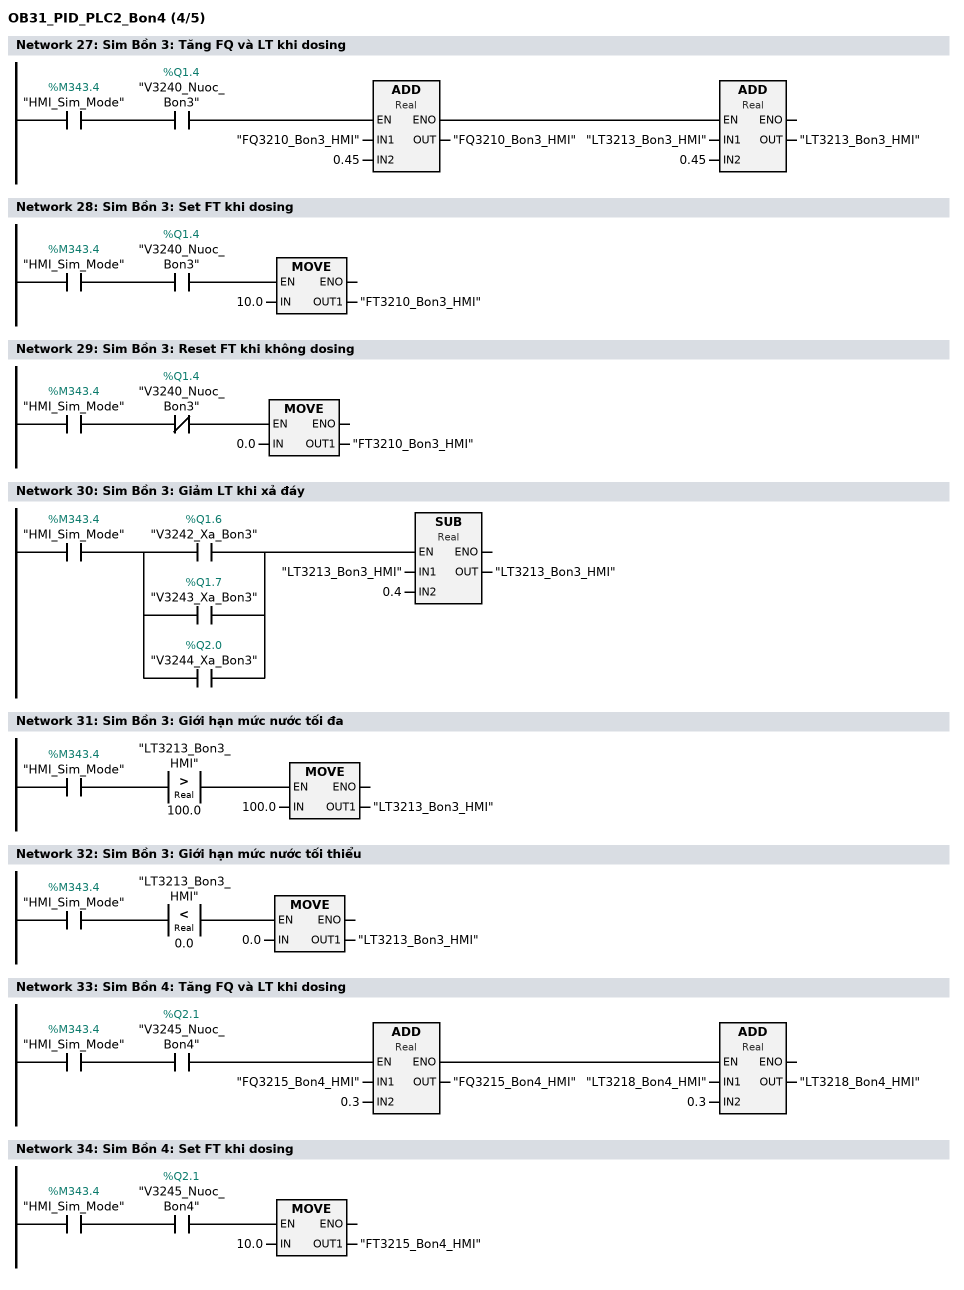
   RUNG wire#powerrail
      Contact( "HMI_Sim_Mode" )
      Contact( "V3240_Nuoc_Bon3" )
      { S7_Templates := "SrcType := Real"; S7_GenerateENO := "TRUE" } Add(in1 := "FQ3210_Bon3_HMI", in2 := 0.45, out => "FQ3210_Bon3_HMI")
      { S7_Templates := "SrcType := Real"; S7_GenerateENO := "TRUE" } Add(in1 := "LT3213_Bon3_HMI", in2 := 0.45, out => "LT3213_Bon3_HMI")
   END_RUNG
   // the same network as SCL:
   // ENO of a box is taken as its EN; it also drops when the box reports an error
   IF "HMI_Sim_Mode" AND "V3240_Nuoc_Bon3" THEN
       "FQ3210_Bon3_HMI" := "FQ3210_Bon3_HMI" + 0.45;
       "LT3213_Bon3_HMI" := "LT3213_Bon3_HMI" + 0.45;
   END_IF;
END_REGION

REGION Network 28: Sim Bồn 3: Set FT khi dosing
   RUNG wire#powerrail
      Contact( "HMI_Sim_Mode" )
      Contact( "V3240_Nuoc_Bon3" )
      { S7_GenerateENO := "TRUE" } Move(in := 10.0, out1 => "FT3210_Bon3_HMI")
   END_RUNG
   // the same network as SCL:
   IF "HMI_Sim_Mode" AND "V3240_Nuoc_Bon3" THEN "FT3210_Bon3_HMI" := 10.0; END_IF;
END_REGION

REGION Network 29: Sim Bồn 3: Reset FT khi không dosing
   RUNG wire#powerrail
      Contact( "HMI_Sim_Mode" )
      I_Contact( "V3240_Nuoc_Bon3" )
      { S7_GenerateENO := "TRUE" } Move(in := 0.0, out1 => "FT3210_Bon3_HMI")
   END_RUNG
   // the same network as SCL:
   IF "HMI_Sim_Mode" AND NOT "V3240_Nuoc_Bon3" THEN "FT3210_Bon3_HMI" := 0.0; END_IF;
END_REGION

REGION Network 30: Sim Bồn 3: Giảm LT khi xả đáy
   RUNG wire#powerrail
      Contact( "HMI_Sim_Mode" )
      wire#w1
      Contact( "V3242_Xa_Bon3" )
      wire#w2
      { S7_Templates := "SrcType := Real"; S7_GenerateENO := "TRUE" } Sub(in1 := "LT3213_Bon3_HMI", in2 := 0.4, out => "LT3213_Bon3_HMI")
   END_RUNG
   RUNG wire#w1
      Contact( "V3243_Xa_Bon3" )
   END_RUNG wire#w2
   RUNG wire#w1
      Contact( "V3244_Xa_Bon3" )
   END_RUNG wire#w2
   // the same network as SCL:
   IF "HMI_Sim_Mode" AND ("V3242_Xa_Bon3" OR "V3243_Xa_Bon3" OR "V3244_Xa_Bon3") THEN
       "LT3213_Bon3_HMI" := "LT3213_Bon3_HMI" - 0.4;
   END_IF;
END_REGION

REGION Network 31: Sim Bồn 3: Giới hạn mức nước tối đa
   RUNG wire#powerrail
      Contact( "HMI_Sim_Mode" )
      { S7_Templates := "SrcType := Real" } GT_Contact(in1 := "LT3213_Bon3_HMI", in2 := 100.0)
      { S7_GenerateENO := "TRUE" } Move(in := 100.0, out1 => "LT3213_Bon3_HMI")
   END_RUNG
   // the same network as SCL:
   IF "HMI_Sim_Mode" AND ("LT3213_Bon3_HMI" > 100.0) THEN "LT3213_Bon3_HMI" := 100.0; END_IF;
END_REGION

REGION Network 32: Sim Bồn 3: Giới hạn mức nước tối thiểu
   RUNG wire#powerrail
      Contact( "HMI_Sim_Mode" )
      { S7_Templates := "SrcType := Real" } LT_Contact(in1 := "LT3213_Bon3_HMI", in2 := 0.0)
      { S7_GenerateENO := "TRUE" } Move(in := 0.0, out1 => "LT3213_Bon3_HMI")
   END_RUNG
   // the same network as SCL:
   IF "HMI_Sim_Mode" AND ("LT3213_Bon3_HMI" < 0.0) THEN "LT3213_Bon3_HMI" := 0.0; END_IF;
END_REGION

REGION Network 33: Sim Bồn 4: Tăng FQ và LT khi dosing
   RUNG wire#powerrail
      Contact( "HMI_Sim_Mode" )
      Contact( "V3245_Nuoc_Bon4" )
      { S7_Templates := "SrcType := Real"; S7_GenerateENO := "TRUE" } Add(in1 := "FQ3215_Bon4_HMI", in2 := 0.3, out => "FQ3215_Bon4_HMI")
      { S7_Templates := "SrcType := Real"; S7_GenerateENO := "TRUE" } Add(in1 := "LT3218_Bon4_HMI", in2 := 0.3, out => "LT3218_Bon4_HMI")
   END_RUNG
   // the same network as SCL:
   // ENO of a box is taken as its EN; it also drops when the box reports an error
   IF "HMI_Sim_Mode" AND "V3245_Nuoc_Bon4" THEN
       "FQ3215_Bon4_HMI" := "FQ3215_Bon4_HMI" + 0.3;
       "LT3218_Bon4_HMI" := "LT3218_Bon4_HMI" + 0.3;
   END_IF;
END_REGION

REGION Network 34: Sim Bồn 4: Set FT khi dosing
   RUNG wire#powerrail
      Contact( "HMI_Sim_Mode" )
      Contact( "V3245_Nuoc_Bon4" )
      { S7_GenerateENO := "TRUE" } Move(in := 10.0, out1 => "FT3215_Bon4_HMI")
   END_RUNG
   // the same network as SCL:
   IF "HMI_Sim_Mode" AND "V3245_Nuoc_Bon4" THEN "FT3215_Bon4_HMI" := 10.0; END_IF;
END_REGION

REGION Network 35: Sim Bồn 4: Reset FT khi không dosing
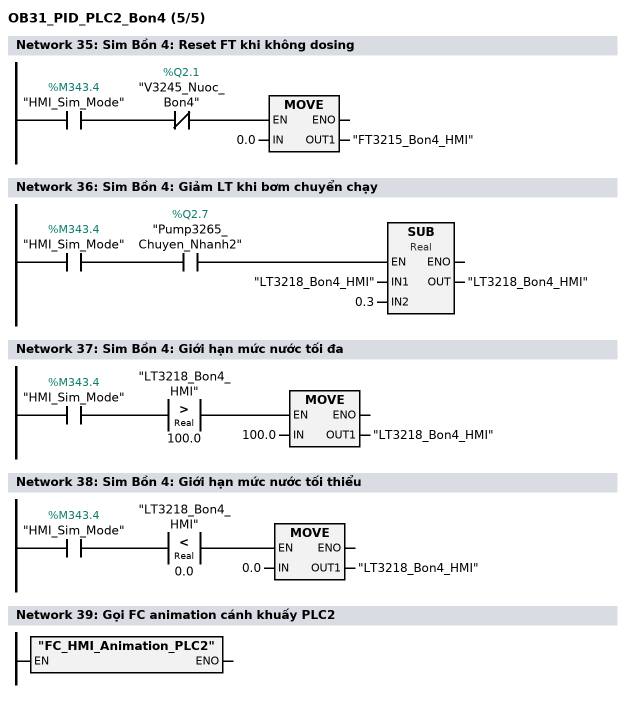
   RUNG wire#powerrail
      Contact( "HMI_Sim_Mode" )
      I_Contact( "V3245_Nuoc_Bon4" )
      { S7_GenerateENO := "TRUE" } Move(in := 0.0, out1 => "FT3215_Bon4_HMI")
   END_RUNG
   // the same network as SCL:
   IF "HMI_Sim_Mode" AND NOT "V3245_Nuoc_Bon4" THEN "FT3215_Bon4_HMI" := 0.0; END_IF;
END_REGION

REGION Network 36: Sim Bồn 4: Giảm LT khi bơm chuyển chạy
   RUNG wire#powerrail
      Contact( "HMI_Sim_Mode" )
      Contact( "Pump3265_Chuyen_Nhanh2" )
      { S7_Templates := "SrcType := Real"; S7_GenerateENO := "TRUE" } Sub(in1 := "LT3218_Bon4_HMI", in2 := 0.3, out => "LT3218_Bon4_HMI")
   END_RUNG
   // the same network as SCL:
   IF "HMI_Sim_Mode" AND "Pump3265_Chuyen_Nhanh2" THEN "LT3218_Bon4_HMI" := "LT3218_Bon4_HMI" - 0.3; END_IF;
END_REGION

REGION Network 37: Sim Bồn 4: Giới hạn mức nước tối đa
   RUNG wire#powerrail
      Contact( "HMI_Sim_Mode" )
      { S7_Templates := "SrcType := Real" } GT_Contact(in1 := "LT3218_Bon4_HMI", in2 := 100.0)
      { S7_GenerateENO := "TRUE" } Move(in := 100.0, out1 => "LT3218_Bon4_HMI")
   END_RUNG
   // the same network as SCL:
   IF "HMI_Sim_Mode" AND ("LT3218_Bon4_HMI" > 100.0) THEN "LT3218_Bon4_HMI" := 100.0; END_IF;
END_REGION

REGION Network 38: Sim Bồn 4: Giới hạn mức nước tối thiểu
   RUNG wire#powerrail
      Contact( "HMI_Sim_Mode" )
      { S7_Templates := "SrcType := Real" } LT_Contact(in1 := "LT3218_Bon4_HMI", in2 := 0.0)
      { S7_GenerateENO := "TRUE" } Move(in := 0.0, out1 => "LT3218_Bon4_HMI")
   END_RUNG
   // the same network as SCL:
   IF "HMI_Sim_Mode" AND ("LT3218_Bon4_HMI" < 0.0) THEN "LT3218_Bon4_HMI" := 0.0; END_IF;
END_REGION

REGION Network 39: Gọi FC animation cánh khuấy PLC2
   RUNG wire#powerrail
      "FC_HMI_Animation_PLC2"()
   END_RUNG
   // the same network as SCL:
   "FC_HMI_Animation_PLC2"();
END_REGION
END_ORGANIZATION_BLOCK

FUNCTION "FC_HMI_Animation_PLC2" : Void   // FC61, LAD
{ S7_Optimized_Access := 'TRUE' }
VERSION : 0.1
// stored: AutoNumber true, IsIECCheckEnabled false, SetENOAutomatically false, UDAEnableTagReadback false
BEGIN

REGION Network 1: Cánh khuấy Bồn 3: Tăng khung hình khi chạy
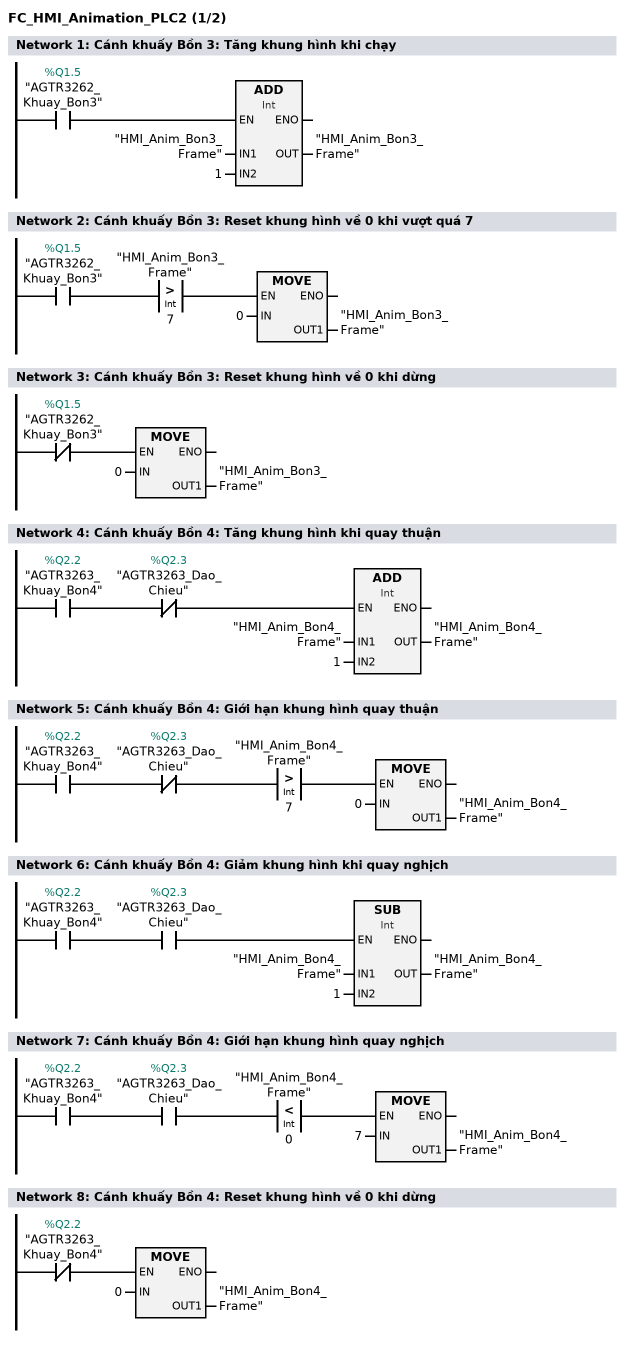
   RUNG wire#powerrail
      Contact( "AGTR3262_Khuay_Bon3" )
      { S7_Templates := "SrcType := Int"; S7_GenerateENO := "TRUE" } Add(in1 := "HMI_Anim_Bon3_Frame", in2 := 1, out => "HMI_Anim_Bon3_Frame")
   END_RUNG
   // the same network as SCL:
   IF "AGTR3262_Khuay_Bon3" THEN "HMI_Anim_Bon3_Frame" := "HMI_Anim_Bon3_Frame" + 1; END_IF;
END_REGION

REGION Network 2: Cánh khuấy Bồn 3: Reset khung hình về 0 khi vượt quá 7
   RUNG wire#powerrail
      Contact( "AGTR3262_Khuay_Bon3" )
      { S7_Templates := "SrcType := Int" } GT_Contact(in1 := "HMI_Anim_Bon3_Frame", in2 := 7)
      { S7_GenerateENO := "TRUE" } Move(in := 0, out1 => "HMI_Anim_Bon3_Frame")
   END_RUNG
   // the same network as SCL:
   IF "AGTR3262_Khuay_Bon3" AND ("HMI_Anim_Bon3_Frame" > 7) THEN "HMI_Anim_Bon3_Frame" := 0; END_IF;
END_REGION

REGION Network 3: Cánh khuấy Bồn 3: Reset khung hình về 0 khi dừng
   RUNG wire#powerrail
      I_Contact( "AGTR3262_Khuay_Bon3" )
      { S7_GenerateENO := "TRUE" } Move(in := 0, out1 => "HMI_Anim_Bon3_Frame")
   END_RUNG
   // the same network as SCL:
   IF NOT "AGTR3262_Khuay_Bon3" THEN "HMI_Anim_Bon3_Frame" := 0; END_IF;
END_REGION

REGION Network 4: Cánh khuấy Bồn 4: Tăng khung hình khi quay thuận
   RUNG wire#powerrail
      Contact( "AGTR3263_Khuay_Bon4" )
      I_Contact( "AGTR3263_Dao_Chieu" )
      { S7_Templates := "SrcType := Int"; S7_GenerateENO := "TRUE" } Add(in1 := "HMI_Anim_Bon4_Frame", in2 := 1, out => "HMI_Anim_Bon4_Frame")
   END_RUNG
   // the same network as SCL:
   IF "AGTR3263_Khuay_Bon4" AND NOT "AGTR3263_Dao_Chieu" THEN
       "HMI_Anim_Bon4_Frame" := "HMI_Anim_Bon4_Frame" + 1;
   END_IF;
END_REGION

REGION Network 5: Cánh khuấy Bồn 4: Giới hạn khung hình quay thuận
   RUNG wire#powerrail
      Contact( "AGTR3263_Khuay_Bon4" )
      I_Contact( "AGTR3263_Dao_Chieu" )
      { S7_Templates := "SrcType := Int" } GT_Contact(in1 := "HMI_Anim_Bon4_Frame", in2 := 7)
      { S7_GenerateENO := "TRUE" } Move(in := 0, out1 => "HMI_Anim_Bon4_Frame")
   END_RUNG
   // the same network as SCL:
   IF "AGTR3263_Khuay_Bon4" AND NOT "AGTR3263_Dao_Chieu" AND ("HMI_Anim_Bon4_Frame" > 7) THEN
       "HMI_Anim_Bon4_Frame" := 0;
   END_IF;
END_REGION

REGION Network 6: Cánh khuấy Bồn 4: Giảm khung hình khi quay nghịch
   RUNG wire#powerrail
      Contact( "AGTR3263_Khuay_Bon4" )
      Contact( "AGTR3263_Dao_Chieu" )
      { S7_Templates := "SrcType := Int"; S7_GenerateENO := "TRUE" } Sub(in1 := "HMI_Anim_Bon4_Frame", in2 := 1, out => "HMI_Anim_Bon4_Frame")
   END_RUNG
   // the same network as SCL:
   IF "AGTR3263_Khuay_Bon4" AND "AGTR3263_Dao_Chieu" THEN
       "HMI_Anim_Bon4_Frame" := "HMI_Anim_Bon4_Frame" - 1;
   END_IF;
END_REGION

REGION Network 7: Cánh khuấy Bồn 4: Giới hạn khung hình quay nghịch
   RUNG wire#powerrail
      Contact( "AGTR3263_Khuay_Bon4" )
      Contact( "AGTR3263_Dao_Chieu" )
      { S7_Templates := "SrcType := Int" } LT_Contact(in1 := "HMI_Anim_Bon4_Frame", in2 := 0)
      { S7_GenerateENO := "TRUE" } Move(in := 7, out1 => "HMI_Anim_Bon4_Frame")
   END_RUNG
   // the same network as SCL:
   IF "AGTR3263_Khuay_Bon4" AND "AGTR3263_Dao_Chieu" AND ("HMI_Anim_Bon4_Frame" < 0) THEN
       "HMI_Anim_Bon4_Frame" := 7;
   END_IF;
END_REGION

REGION Network 8: Cánh khuấy Bồn 4: Reset khung hình về 0 khi dừng
   RUNG wire#powerrail
      I_Contact( "AGTR3263_Khuay_Bon4" )
      { S7_GenerateENO := "TRUE" } Move(in := 0, out1 => "HMI_Anim_Bon4_Frame")
   END_RUNG
   // the same network as SCL:
   IF NOT "AGTR3263_Khuay_Bon4" THEN "HMI_Anim_Bon4_Frame" := 0; END_IF;
END_REGION

REGION Network 9: Bồn 3 Mức dịch: Rỗng khi LT <= 0.5
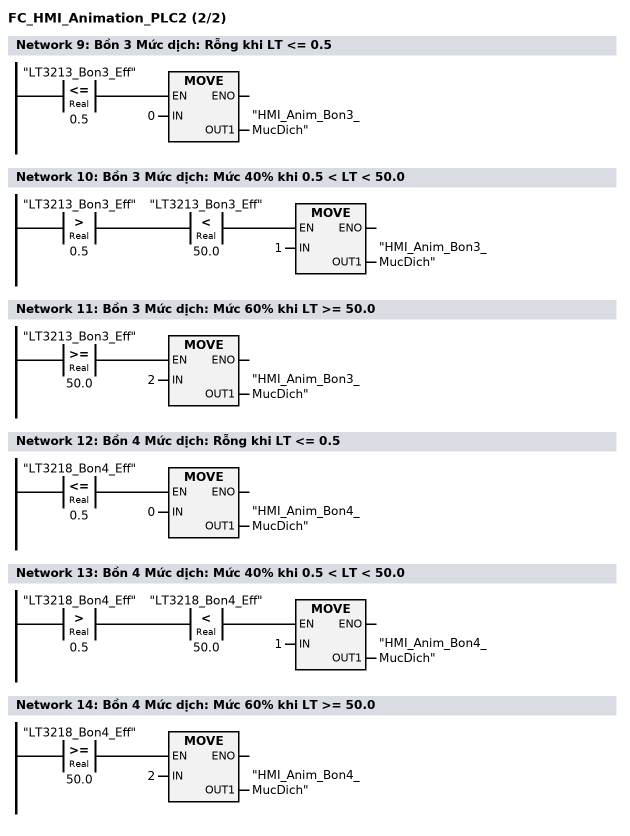
   RUNG wire#powerrail
      { S7_Templates := "SrcType := Real" } LE_Contact(in1 := "LT3213_Bon3_Eff", in2 := 0.5)
      { S7_GenerateENO := "TRUE" } Move(in := 0, out1 => "HMI_Anim_Bon3_MucDich")
   END_RUNG
   // the same network as SCL:
   IF "LT3213_Bon3_Eff" <= 0.5 THEN "HMI_Anim_Bon3_MucDich" := 0; END_IF;
END_REGION

REGION Network 10: Bồn 3 Mức dịch: Mức 40% khi 0.5 < LT < 50.0
   RUNG wire#powerrail
      { S7_Templates := "SrcType := Real" } GT_Contact(in1 := "LT3213_Bon3_Eff", in2 := 0.5)
      { S7_Templates := "SrcType := Real" } LT_Contact(in1 := "LT3213_Bon3_Eff", in2 := 50.0)
      { S7_GenerateENO := "TRUE" } Move(in := 1, out1 => "HMI_Anim_Bon3_MucDich")
   END_RUNG
   // the same network as SCL:
   IF ("LT3213_Bon3_Eff" > 0.5) AND ("LT3213_Bon3_Eff" < 50.0) THEN "HMI_Anim_Bon3_MucDich" := 1; END_IF;
END_REGION

REGION Network 11: Bồn 3 Mức dịch: Mức 60% khi LT >= 50.0
   RUNG wire#powerrail
      { S7_Templates := "SrcType := Real" } GE_Contact(in1 := "LT3213_Bon3_Eff", in2 := 50.0)
      { S7_GenerateENO := "TRUE" } Move(in := 2, out1 => "HMI_Anim_Bon3_MucDich")
   END_RUNG
   // the same network as SCL:
   IF "LT3213_Bon3_Eff" >= 50.0 THEN "HMI_Anim_Bon3_MucDich" := 2; END_IF;
END_REGION

REGION Network 12: Bồn 4 Mức dịch: Rỗng khi LT <= 0.5
   RUNG wire#powerrail
      { S7_Templates := "SrcType := Real" } LE_Contact(in1 := "LT3218_Bon4_Eff", in2 := 0.5)
      { S7_GenerateENO := "TRUE" } Move(in := 0, out1 => "HMI_Anim_Bon4_MucDich")
   END_RUNG
   // the same network as SCL:
   IF "LT3218_Bon4_Eff" <= 0.5 THEN "HMI_Anim_Bon4_MucDich" := 0; END_IF;
END_REGION

REGION Network 13: Bồn 4 Mức dịch: Mức 40% khi 0.5 < LT < 50.0
   RUNG wire#powerrail
      { S7_Templates := "SrcType := Real" } GT_Contact(in1 := "LT3218_Bon4_Eff", in2 := 0.5)
      { S7_Templates := "SrcType := Real" } LT_Contact(in1 := "LT3218_Bon4_Eff", in2 := 50.0)
      { S7_GenerateENO := "TRUE" } Move(in := 1, out1 => "HMI_Anim_Bon4_MucDich")
   END_RUNG
   // the same network as SCL:
   IF ("LT3218_Bon4_Eff" > 0.5) AND ("LT3218_Bon4_Eff" < 50.0) THEN "HMI_Anim_Bon4_MucDich" := 1; END_IF;
END_REGION

REGION Network 14: Bồn 4 Mức dịch: Mức 60% khi LT >= 50.0
   RUNG wire#powerrail
      { S7_Templates := "SrcType := Real" } GE_Contact(in1 := "LT3218_Bon4_Eff", in2 := 50.0)
      { S7_GenerateENO := "TRUE" } Move(in := 2, out1 => "HMI_Anim_Bon4_MucDich")
   END_RUNG
   // the same network as SCL:
   IF "LT3218_Bon4_Eff" >= 50.0 THEN "HMI_Anim_Bon4_MucDich" := 2; END_IF;
END_REGION
END_FUNCTION
